PROGRAM MAIN
VAR
END_VAR

END_PROGRAM

(* stored: Version 1.1.0.1
   POU MAIN: Id {77ce3c58-9155-42f5-9eb6-c02febfddbf9} *)
